(* CODESYS project Aufzug20.project

Project tree, tasks and I/O mapping:
  Device : CODESYS Control Win V3, 3S - Smart Software Solutions GmbH, order no. 305021, version 3.5.10.60
    application Application
      libraries: Standard, * (System); Util, * (System)
      task VISU_TASK (cyclic, interval 100 ms, priority 31) calls VisuElems.Visu_Prg
      task MainTask (cyclic, interval t#20ms, priority 1) calls PLC_PRG
      function block ManualControl [ST]
      data type Sensors
      global variables GVL_HMI
      global variables GVL_KONSTANTEN
      global variables GVL_AUFZUG
      Symbols
      program PLC_PRG [ST]
      function block OperatingMode [ST]
      visualisation Visualization
      function block DoorControl [ST]
      function SpeedCalculation [ST]
      function block Position [ST]
      function block MotorControl [ST]
      function block AuftragsTest [ST]
      data type Level
      function block LevelAnfahren [ST]
      function CalculateDirection [ST]
      function block Auftragsmanager [ST]
    Ethernet : Ethernet, 3S - Smart Software Solutions GmbH, version 3.5.10.0
        settings: IPAddress = [141,37,200,19]; SubnetMask = [255,255,255,255]; GatewayAddress = [0,0,0,0]; MACAddress = [16#00,16#00,16#00,16#00,16#00,16#00]; NetworkInterfaceName = 'htwg'; NetworkInterfaceName = "htwg"; SaveCommunicationSettings = FALSE
      Modbus_TCP_Master : Modbus TCP Master, 3S - Smart Software Solutions GmbH, version 3.5.10.0
        Modbus_TCP_Slave : Modbus TCP Slave, 3S - Smart Software Solutions GmbH, version 3.5.10.0
            settings: IPAddress = [141, 37, 159, 111]; Port = 503; Channel 0.Function Code = 4; Channel 0.Read Offset = 16#0000; Channel 0.Read Length = 7; Channel 0.Write Offset = 0; Channel 0.Write Length = 0; Channel 0.Cycle Time = 100; Channel 1.Function Code = 16; Channel 1.Read Offset = 0; Channel 1.Read Length = 0; Channel 1.Write Offset = 16#0000; Channel 1.Write Length = 2; Channel 1.Cycle Time = 100
            unmapped channels: Channel 0, Channel 1
  text list GlobalTextList
*)

// Device/Application/Sensors
TYPE Sensors :
STRUCT
	approach_lower :BOOL;
	safety_lower :BOOL;
	reached :BOOL;
	safety_upper :BOOL;
	approach_upper :BOOL;
END_STRUCT
END_TYPE

// Device/Application/Level
TYPE Level :
STRUCT
	sensors : Sensors;
	anforderungNachOben	: BOOL;
	anforderungNachUnten : BOOL;
END_STRUCT
END_TYPE

// Device/Application/GVL_HMI
{attribute 'qualified_only'}
VAR_GLOBAL
	//------------------------------------------------------------------------------------
	// Buttons
		// Operator								Taster die der Operator und Supervisor siehr
		Button_DoorClose			:BOOL;		// Taster innen Anforderung Tür schließen
		Button_DoorOpen				:BOOL;		// Taster innen Anforderung Türe Öffnen
		Button_EmergencyStop		:BOOL;		// Taster innen Anforderung Nothalt
		Buttons_level				:ARRAY[GVL_KONSTANTEN.min_level..GVL_KONSTANTEN.max_level] OF BOOL;
												// Taster innen Anforderung der Level (In unserem Fall Level 1,2,3,4)
		Buttons_Up					:ARRAY[GVL_KONSTANTEN.min_level..(GVL_KONSTANTEN.max_level-1)] OF BOOL;
												// Taster außen Anforderung Hochfahren (In unserem Fall Level 1,2,3)
		Buttons_Down				:ARRAY[(GVL_KONSTANTEN.min_level+1)..GVL_KONSTANTEN.max_level] OF BOOL;
												// Taster außen Anforderung Runterfahren (In unserem Fall Level 2,3,4)
												
		// Supervisor							Taster die der Supervisor zusätzlich hat
		Button_Reset				:BOOL;		// Taster Simulation-Reset
		Button_DoorCloseManual		:BOOL;		// Taster Handbetrieb Türe schließen
		Button_DoorOpenManual		:BOOL;		// Taster Handbetrieb Türe öffnen
		Button_MotorUpV1Manual		:BOOL;		// Taster Handbetrieb hochfahren mit V1
		Button_MotorUpV2Manual		:BOOL;		// Taster Handbetrieb hochfahren mit V2
		Button_MotorUpCrawlManual	:BOOL;		// Taster Handbetrieb hochfahren mit Kriechgeschwindigkeit
		Button_MotorDownV1Manual	:BOOL;		// Taster Handbetrieb runterfahren mit V1
		Button_MotorDownV2Manual	:BOOL;		// Taster Handbetrieb runterfahren mit V2
		Button_MotorDownCrawlManual	:BOOL;		// Taster Handbetrieb runterfahren mit Kriechgeschwindigkeit
		Button_AutomaticMode		:BOOL;		// Taster Anforderung Automatikmodus
		Button_ManualMode			:BOOL;		// Taster Anforderung Handbetrieb
		
		Button_deleteRequests		:BOOL;
		
		SupervisorActive			:BOOL;		// Variable Benutzerebenen
		
	//------------------------------------------------------------------------------------
	// Anzeigen
		ErrorState					:BOOL;		// Anzeige Aufzug befindet sich in Fehlerzustand
		
		DoorOpens					:BOOL;		// Anzeige Türe öffnet sich
		DoorCloses					:BOOL; 		// Anzeige Türe schließt sich
		DoorIsOpen					:BOOL;		// Anzeige Türe ist offen
		DoorIsClosed				:BOOL;		// Anzeige Türe ist geschlossen
		
		SimulationDoorIsOpen		:ARRAY[GVL_KONSTANTEN.min_level..GVL_KONSTANTEN.max_level] OF BOOL;
												// Simulation, welche Türe in welcher Etage offen ist
		
		AutomaticMode				:BOOL;		// Anzeige Automatikmodus
		ManualMode					:BOOL;		// Anzeige Handbetrieb
		
		MotorReady					:BOOL;		// Anzeige Motor ist bereit
		MotorOn						:BOOL;		// Anzeige Motor läuft
		MotorUp						:BOOL;		// Anzeige Aufzug fährt nach oben
		MotorDown					:BOOL;		// Anzeige Aufzug fährt nach unten
		MotorUpV1					:BOOL;		// Anzeige Aufzug fährt nach oben mit V1
		MotorUpV2					:BOOL;		// Anzeige Aufzug fährt nach oben mit V2
		MotorUpCrawl				:BOOL;		// Anzeige Aufzug fährt nach oben mit Kriechgeschwindigkeit
		MotorDownV1					:BOOL;		// Anzeige Aufzug fährt nach unten mit V1
		MotorDownV2					:BOOL;		// Anzeige Aufzug fährt nach unten mit V2
		MotorDownCrawl				:BOOL;		// Anzeige Aufzug fährt nach unten mit Kriechgeschwindigkeit
		Speed						:REAL;		// Anzeige akturelle Geschwindigkeit in m/s
		
		CurrentLevel				:INT;		// Anzeige in welchem Level sich der Aufzug gerade befindet
		TargetLevel					:INT;		// Anzeige, des aktuellen ZielStockwerks
		
		Requests					:ARRAY[GVL_KONSTANTEN.min_level..GVL_KONSTANTEN.max_level, 1..3] OF BOOL;
												// Anzeigen welche Stockwerke angefordert werden
		Sensors						:ARRAY[GVL_KONSTANTEN.min_level..GVL_KONSTANTEN.max_level, 1..5] OF BOOL;
												// Anzeige aktiver Sensoren
		LevelArrival				:ARRAY[GVL_KONSTANTEN.min_level..GVL_KONSTANTEN.max_level] OF BOOL;
		LevelDeparture				:ARRAY[GVL_KONSTANTEN.min_level..GVL_KONSTANTEN.max_level] OF BOOL;
		Position					:INT;		// Anzeige Aufzugsposition in mm
		
												
END_VAR

// Device/Application/GVL_KONSTANTEN
{attribute 'qualified_only'}
VAR_GLOBAL CONSTANT
	min_level	:INT:=1;
	max_level	:INT:=4;
	
	holding_period	:TIME:=T#6S;
END_VAR

// Device/Application/GVL_AUFZUG
{attribute 'qualified_only'}
VAR_GLOBAL
	// Ausgänge
	POreset 			AT %QX0.0 : BOOL; 		// Simulation reset
	POdv2 				AT %QX1.0 : BOOL; 		// motor setpoint down v2
	POdv1 				AT %QX1.1 : BOOL; 		// motor setpoint down v1
	POuv1 				AT %QX1.2 : BOOL; 		// motor setpoint up v1
	POuv2 				AT %QX1.3 : BOOL; 		// motor setpoint up v2
	POdclose 			AT %QX1.4 : BOOL; 		// motor close door
	POdopen 			AT %QX1.5 : BOOL; 		// motor open door
	POv_crawlSelect 	AT %QW1 : INT (-5..5); 	// select crawl speed; -5..5 cm/s
	
	// Eingänge
	PIs_l1sl 			AT %IX0.1 : BOOL; 		// Level 1 safety lower
	PIs_l1r 			AT %IX0.2 : BOOL; 		// Level 1 reached
	PIs_l1su 			AT %IX0.3 : BOOL; 		// Level 1 safety upper
	PIs_l1au 			AT %IX0.4 : BOOL; 		// Level 1 approach upper
	PIs_l2al 			AT %IX1.0 : BOOL; 		// Level 2 approach lower
	PIs_l2sl 			AT %IX1.1 : BOOL; 		// etc.
	PIs_l2r 			AT %IX1.2 : BOOL;
	PIs_l2su 			AT %IX1.3 : BOOL;
	PIs_l2au 			AT %IX1.4 : BOOL;
	PIs_l3al 			AT %IX2.0 : BOOL;
	PIs_l3sl 			AT %IX2.1 : BOOL;
	PIs_l3r 			AT %IX2.2 : BOOL;
	PIs_l3su 			AT %IX2.3 : BOOL;
	PIs_l3au 			AT %IX2.4 : BOOL;
	PIs_l4al 			AT %IX3.0 : BOOL;
	PIs_l4sl 			AT %IX3.1 : BOOL;
	PIs_l4r 			AT %IX3.2 : BOOL;
	PIs_l4su 			AT %IX3.3 : BOOL;
	PIcycles 			AT %ID1 : UDINT; 		// PLC cycles since start
	PIaufzugID 			AT %IW4 : UINT; 		// instance identifier (1..4)
	PIs_dopened 		AT %IX10.0 : BOOL; 		// door is open
	PIs_dclosed 		AT %IX10.1 : BOOL; 		// door is closed
	PIm_ready 			AT %IX10.2 : BOOL; 		// motor ready
	PIm_on 				AT %IX10.3 : BOOL; 		// motor is on
	PIm_error 			AT %IX10.4 : BOOL; 		// error state; reset with POreset
	PIs_v 				AT %IW6 : INT; 			// v [v]=1cm/s
END_VAR

// Device/Application/PLC_PRG
PROGRAM PLC_PRG
VAR	
	levels : ARRAY[GVL_KONSTANTEN.min_level..GVL_KONSTANTEN.max_level] OF Level;
	
	// FB Instanzen
	betriebsart			:OperatingMode;
	handBetrieb			:ManualControl;
	tuere  				: DoorControl;
	position 			: Position;
	motorControl 		: MotorControl;
	auftrag				: AuftragsTest;
	auftragsmanager		: Auftragsmanager;
	
	// Schnittstellen Funktionsbausteine
	automatik_ein				: BOOL;
	handbetrieb_ein				: BOOL;
	elevator_in_reached_position	: BOOL;
	level_target				: INT;
	level_current				: INT;
	level_target_reached		: BOOL;
	waiting_for_request			: BOOL;
	request_door_aut			: BOOL;

	// Zähler
	i : INT;
	
END_VAR

// Initialisierung Array
levels[GVL_KONSTANTEN.min_level].sensors.approach_lower		:= FALSE;
levels[GVL_KONSTANTEN.min_level].sensors.safety_lower		:= GVL_AUFZUG.PIs_l1sl;
levels[GVL_KONSTANTEN.min_level].sensors.reached			:= GVL_AUFZUG.PIs_l1r;
levels[GVL_KONSTANTEN.min_level].sensors.safety_upper		:= GVL_AUFZUG.PIs_l1su;
levels[GVL_KONSTANTEN.min_level].sensors.approach_upper		:= GVL_AUFZUG.PIs_l1au;
levels[GVL_KONSTANTEN.min_level].anforderungNachUnten		:= FALSE;
levels[GVL_KONSTANTEN.min_level].anforderungNachOben		:= GVL_HMI.Buttons_Up[GVL_KONSTANTEN.min_level];

levels[2].sensors.approach_lower							:= GVL_AUFZUG.PIs_l2al;
levels[2].sensors.safety_lower								:= GVL_AUFZUG.PIs_l2sl;
levels[2].sensors.reached									:= GVL_AUFZUG.PIs_l2r;
levels[2].sensors.safety_upper								:= GVL_AUFZUG.PIs_l2su;
levels[2].sensors.approach_upper							:= GVL_AUFZUG.PIs_l2au;
levels[2].anforderungNachUnten								:= GVL_HMI.Buttons_Down[2];
levels[2].anforderungNachOben								:= GVL_HMI.Buttons_Up[2];

levels[3].sensors.approach_lower							:= GVL_AUFZUG.PIs_l3al;
levels[3].sensors.safety_lower								:= GVL_AUFZUG.PIs_l3sl;
levels[3].sensors.reached									:= GVL_AUFZUG.PIs_l3r;
levels[3].sensors.safety_upper								:= GVL_AUFZUG.PIs_l3su;
levels[3].sensors.approach_upper							:= GVL_AUFZUG.PIs_l3au;
levels[3].anforderungNachUnten								:= GVL_HMI.Buttons_Down[3];
levels[3].anforderungNachOben								:= GVL_HMI.Buttons_Up[3];

levels[GVL_KONSTANTEN.max_level].sensors.approach_lower		:= GVL_AUFZUG.PIs_l4al;
levels[GVL_KONSTANTEN.max_level].sensors.safety_lower		:= GVL_AUFZUG.PIs_l4sl;
levels[GVL_KONSTANTEN.max_level].sensors.reached			:= GVL_AUFZUG.PIs_l4r;
levels[GVL_KONSTANTEN.max_level].sensors.safety_upper		:= GVL_AUFZUG.PIs_l4su;
levels[GVL_KONSTANTEN.max_level].sensors.approach_upper		:= FALSE;
levels[GVL_KONSTANTEN.max_level].anforderungNachUnten		:= GVL_HMI.Buttons_Down[GVL_KONSTANTEN.max_level];
levels[GVL_KONSTANTEN.max_level].anforderungNachOben		:= FALSE;

//------------------------------------------------------------------------------------
// Funktionsbausteine 

// Betriebsart 
betriebsart(
	wechsel_in_automatik := PLC_PRG.elevator_in_reached_position
	);
	
	automatik_ein:= PLC_PRG.betriebsart.automatikBetrieb;
	handbetrieb_ein:= PLC_PRG.betriebsart.handBetrieb;


// Handbetrieb
handBetrieb(
	enableManualControl := PLC_PRG.handbetrieb_ein, 
	freigabe_tuere:= PLC_PRG.elevator_in_reached_position
	);

// Positionsauswertung
position(
	levels:= PLC_PRG.levels
	);
	
	PLC_PRG.elevator_in_reached_position := position.elevator_in_reached_positon;
	PLC_PRG.level_current := position.level_current;

// Motorsteuerung Aufzug	
motorControl(
	automatic_mode := PLC_PRG.automatik_ein,
	levels := PLC_PRG.levels,
	reset := GVL_HMI.Button_Reset,
	level_target := PLC_PRG.level_target,
	level_current := PLC_PRG.level_current,
	emergency_stop := GVL_HMI.Button_EmergencyStop,
	request_DoorControl_start := GVL_HMI.Button_DoorOpen OR PLC_PRG.request_door_aut
	);
	
	PLC_PRG.waiting_for_request := motorControl.waiting_for_request;
	PLC_PRG.level_target_reached := motorControl.next_level_reached;

// Auftragsverarbeitung
auftrag(
	neuen_Auftrag_annehmen:= PLC_PRG.waiting_for_request
	);
	
	//level_target := auftrag.zielstockwerk;

// Auftragsmanager
auftragsmanager(
	levels := PLC_PRG.levels,
	buttons_inside := GVL_HMI.Buttons_level,
	level_current := PLC_PRG.level_current,
	level_target_reached := PLC_PRG.level_target_reached,
	waiting_for_request := PLC_PRG.waiting_for_request,
	request_door_aut	:= ,
	reset				:= GVL_HMI.Button_Reset
	);
	
	PLC_PRG.request_door_aut := auftragsmanager.request_door_aut;
	PLC_PRG.level_target := auftragsmanager.level_target;

// Ausgänge HMI - Anzeigen, Simulationen
GVL_HMI.AutomaticMode := automatik_ein;
GVL_HMI.ManualMode := handbetrieb_ein;

GVL_HMI.ErrorState := GVL_AUFZUG.PIm_error;

GVL_HMI.MotorUpV1 := GVL_AUFZUG.POuv1;
GVL_HMI.MotorUpV2 := GVL_AUFZUG.POuv2;
GVL_HMI.MotorUpCrawl := GVL_AUFZUG.POv_crawlSelect > 0;
GVL_HMI.MotorDownV1 := GVL_AUFZUG.POdv1;
GVL_HMI.MotorDownV2 := GVL_AUFZUG.POdv2;
GVL_HMI.MotorDownCrawl := GVL_AUFZUG.POv_crawlSelect < 0;
GVL_HMI.DoorCloses := GVL_AUFZUG.POdclose;
GVL_HMI.DoorOpens := GVL_AUFZUG.POdopen;
GVL_HMI.DoorIsClosed := GVL_AUFZUG.PIs_dclosed;
GVL_HMI.DoorIsOpen := GVL_AUFZUG.PIs_dopened;

GVL_HMI.MotorDown := motorControl.aufzug_faehrt_nach_unten;
GVL_HMI.MotorUp := motorControl.aufzug_faehrt_nach_oben;

GVL_HMI.CurrentLevel := level_current;
GVL_HMI.TargetLevel := level_target;

GVL_HMI.Requests := auftragsmanager.requests;
GVL_HMI.LevelArrival := motorControl.levelArrival;
GVL_HMI.LevelDeparture := motorControl.levelDeparture;


GVL_HMI.Speed := SpeedCalculation(GVL_AUFzug.PIs_v);
GVL_HMI.Position := position.position;

FOR i := GVL_KONSTANTEN.min_level TO GVL_KONSTANTEN.max_level BY 1 DO
	GVL_HMI.Sensors[i,1] := levels[i].sensors.approach_lower;
	GVL_HMI.Sensors[i,2] := levels[i].sensors.safety_lower;
	GVL_HMI.Sensors[i,3] := levels[i].sensors.reached;
	GVL_HMI.Sensors[i,4] := levels[i].sensors.safety_upper;
	GVL_HMI.Sensors[i,5] := levels[i].sensors.safety_upper;	
END_FOR

FOR i := GVL_KONSTANTEN.min_level TO GVL_KONSTANTEN.max_level BY 1 DO
	IF GVL_AUFZUG.PIs_dclosed THEN
		GVL_HMI.SimulationDoorIsOpen[i] := FALSE;
	END_IF
END_FOR

IF GVL_AUFZUG.PIs_dopened THEN
	GVL_HMI.SimulationDoorIsOpen[position.level_current] := TRUE;
END_IF

// Ausgänge Aufzug-Simulation
GVL_AUFZUG.POreset := GVL_HMI.Button_Reset;

GVL_AUFZUG.POuv1 := handbetrieb.MotorUpV1 OR motorControl.up_V1;
GVL_AUFZUG.POuv2 := handbetrieb.MotorUpV2 OR motorControl.up_V2;
GVL_AUFZUG.POdv1 := handbetrieb.MotorDownV1 OR motorControl.down_V1;
GVL_AUFZUG.POdv2 := handbetrieb.MotorDownV2 OR motorControl.down_V2;
IF handbetrieb_ein AND NOT automatik_ein THEN
	GVL_AUFZUG.POv_crawlSelect := handbetrieb.MotorCrawlSelect;
ELSIF automatik_ein AND NOT handbetrieb_ein THEN
	GVL_AUFZUG.POv_crawlSelect := motorControl.crawl_select;
END_IF
GVL_AUFZUG.POdopen := handbetrieb.MotorOpenDoor OR motorControl.door_open;
GVL_AUFZUG.POdclose := handbetrieb.MotorCloseDoor OR motorControl.door_close;

END_PROGRAM

// Device/Application/Position
FUNCTION_BLOCK Position
VAR_INPUT
	levels : ARRAY[GVL_KONSTANTEN.min_level..GVL_KONSTANTEN.max_level] OF Level;
END_VAR
VAR_OUTPUT
	elevator_in_reached_positon : BOOL;
	level_current : INT;
	position : INT;
	
	
END_VAR
VAR
	i : INT;
	postion_integral : INT;
	positon_sensor : INT;
	integral : INTEGRAL;
	resetIntegral : BOOL:=TRUE;
END_VAR

// Init
elevator_in_reached_positon := FALSE;

integral(
	IN:= GVL_AUFzug.PIs_v,
	TM:=20,
	RESET:= resetIntegral);

postion_integral := REAL_TO_INT(integral.OUT * 10);

resetIntegral:= FALSE;	

// Schleife
FOR i := GVL_KONSTANTEN.min_level TO GVL_KONSTANTEN.max_level BY 1 DO
	
	IF levels[i].sensors.reached THEN
		elevator_in_reached_positon:=TRUE;
		resetIntegral := TRUE;
		positon_sensor := i*3500 - 3500;
		level_current:= i;
	END_IF
	
	IF levels[i].sensors.approach_lower THEN
		resetIntegral := TRUE;
		positon_sensor := i*3500 - 3500 - 1500;
		level_current:= i;
	END_IF
	
	IF levels[i].sensors.safety_lower THEN
		resetIntegral := TRUE;
		positon_sensor := i*3500 -3500 -50;
		level_current:= i;
	END_IF
	
	IF levels[i].sensors.safety_upper THEN
		resetIntegral := TRUE;
		positon_sensor := i*3500 - 3500 + 50;
		level_current:= i;
	END_IF
	
	IF levels[i].sensors.approach_upper THEN
		resetIntegral := TRUE;
		positon_sensor := i*3500 -3500 + 1500;
		level_current:= i;
	END_IF
	
END_FOR

// Ausgänge
position := positon_sensor + postion_integral;

END_FUNCTION_BLOCK

// Device/Application/MotorControl
FUNCTION_BLOCK MotorControl
VAR_INPUT
	levels 				: ARRAY[GVL_KONSTANTEN.min_level..GVL_KONSTANTEN.max_level] OF Level;
	reset 				: BOOL;
	level_target 		: INT := GVL_KONSTANTEN.min_level;
	level_current 		: INT := GVL_KONSTANTEN.max_level;
	automatic_mode 		: BOOL;
	emergency_stop 		: BOOL;
	request_DoorControl_start 	: BOOL;
END_VAR
VAR_OUTPUT
	up_V1 : BOOL;
	up_V2 : BOOL;
	down_V1 : BOOL;
	down_V2 : BOOL;
	crawl_select : INT;
	door_open : BOOL;
	door_close : BOOL;
	
	waiting_for_request : BOOL;
	next_level_reached : BOOL;
	
	levelArrival				:ARRAY[GVL_KONSTANTEN.min_level..GVL_KONSTANTEN.max_level] OF BOOL;
	levelDeparture				:ARRAY[GVL_KONSTANTEN.min_level..GVL_KONSTANTEN.max_level] OF BOOL;
	
	aufzug_faehrt_nach_oben : BOOL;
	aufzug_faehrt_nach_unten : BOOL;
END_VAR
VAR
	z		: INT:=0;
	
	direction_up : BOOL; 
	direction_down : BOOL;
	
	levelAnfahrenNachOben	: LevelAnfahren;
	levelAnfahrenNachUnten	: LevelAnfahren;
	doorControl : DoorControl;
END_VAR

levelAnfahrenNachOben(
	start := (z=20),
	sensor_reached := levels[level_target].sensors.reached,
	sensor_safty_before := levels[level_target].sensors.safety_lower,
	sensor_safty_after := levels[level_target].sensors.safety_upper,
	sensor_approach := levels[level_target].sensors.approach_lower,
	emergency_stop := emergency_stop,
	reset := reset OR NOT automatic_mode,
	direction_up := TRUE
	);
	
levelAnfahrenNachUnten(
	start := (z=30),
	sensor_reached := levels[level_target].sensors.reached,
	sensor_safty_before := levels[level_target].sensors.safety_upper,
	sensor_safty_after := levels[level_target].sensors.safety_lower,
	sensor_approach := levels[level_target].sensors.approach_upper,
	emergency_stop := emergency_stop,
	reset := reset OR NOT automatic_mode,
	direction_up := FALSE
	);

doorControl(
	aut_start:= z=40
	);

// Gehe in Initialisierungszustand, wenn Reset
IF reset OR NOT automatic_mode THEN
	z:=0;
	direction_up :=FALSE;
	direction_down := FALSE;
END_IF 

// Zustandsautomat
CASE z OF
	// Init, Reset
	0:
	IF GVL_AUFZUG.PIm_ready THEN
		z:=10;
	END_IF
	
	// Wartezustand - Aufzug befindet sich in Ziellevel und wartet auf nächsten Auftrag
	10:
	IF level_target > level_current THEN
		z:=20;
	ELSIF level_target < level_current THEN
		z:= 30;
	END_IF
	
	IF request_DoorControl_start THEN
		z:= 40;
	END_IF
	
	// Impuls nach oben Anfahren
	20:
	z:= 21;
	
	//  Level anfahren
	21:
	IF levelAnfahrenNachOben.level_reached THEN
		z:=40;
	END_IF
	
	// Impuls nach unten Anfahren
	30:
	z:= 31;
	
	// Level Anfahren
	31:
	IF levelAnfahrenNachUnten.level_reached THEN
		z:=40;
	END_IF
	
	// Impuls Türautomatik Start, Level Angefahren
	40:
	z:= 41;
	
	// Warte auf Ende Türautomatik	
	41:
	IF doorControl.aut_ende THEN
		z:=10;
	END_IF
	
END_CASE
	

up_V1 := levelAnfahrenNachOben.v1;
up_V2 := levelAnfahrenNachOben.v2;
down_V1 := levelAnfahrenNachUnten.v1;
down_V2 := levelAnfahrenNachUnten.v2;
door_open := doorControl.door_open;
door_close := doorControl.door_close;

IF levelAnfahrenNachOben.fb_active THEN
	crawl_select := levelAnfahrenNachOben.crawl_select;
ELSIF levelAnfahrenNachUnten.fb_active THEN
	crawl_select := levelAnfahrenNachUnten.crawl_select;
ELSE
	crawl_select := 0;
END_IF

waiting_for_request := z=10 OR z=40 OR z=41;
next_level_reached := z=40;

IF z=10 OR z=40 OR z=41 THEN
	levelArrival[level_current] := TRUE;
ELSE
	levelArrival[level_current] := FALSE;
END_IF
IF z=20 OR z=30 THEN
	levelDeparture[level_current] :=TRUE;
ELSE
	levelDeparture[level_current] :=FALSE;
END_IF

aufzug_faehrt_nach_oben := levelAnfahrenNachOben.fb_active;
aufzug_faehrt_nach_unten := levelAnfahrenNachUnten.fb_active;

END_FUNCTION_BLOCK

// Device/Application/DoorControl
FUNCTION_BLOCK DoorControl
VAR_INPUT
	aut_start : BOOL;
END_VAR
VAR_OUTPUT
	aut_ende :BOOL;
	door_open : BOOL;
	door_close : BOOL;
END_VAR
VAR
	z: INT:=0;
	ton_halten :TON;
	i_max : INT:=3;
END_VAR

ton_halten(IN:=z=3, PT:= T#6S);

CASE z OF
	// Init
	0:
	z:=1;
	
	// Wartezustand
	1:
	IF aut_start  THEN
		z:=2;
		i_max:=3;
	END_IF
	
	// Tuere öffnen
	2:
	IF GVL_AUFZUG.PIs_dopened THEN
		z:=3;
	END_IF
	
	// Tuere offen halten
	3:
	IF ton_halten.Q OR GVL_HMI.Button_DoorCloseManual OR GVL_HMI.Button_DoorClose THEN
		z:=4;
	END_IF
	
	// Tuere schließen
	4:
	IF GVL_AUFZUG.PIs_dclosed THEN
		z:=5;
	END_IF
	IF i_max > 0 AND (GVL_HMI.Button_DoorOpenManual OR GVL_HMI.Button_DoorOpen) THEN			// Türe wieder aufmachen
		z:=2;
		i_max:= i_max - 1;
	END_IF
	
	// Ende
	5:
	z:=0;
END_CASE

// Ausgänge
aut_ende := z=5;
door_open:= z=2;
door_close:= z=4;

END_FUNCTION_BLOCK

// Device/Application/LevelAnfahren
FUNCTION_BLOCK LevelAnfahren
VAR_INPUT
	start 				: BOOL;
	sensor_reached 		: BOOL;
	sensor_safty_before : BOOL;
	sensor_safty_after	: BOOL;
	sensor_approach		: BOOL;
	emergency_stop		: BOOL;
	reset				: BOOL;
	direction_up		: BOOL;
END_VAR
VAR_OUTPUT
	v1	: BOOL;
	v2 	: BOOL;
	crawl_select	: INT :=0;
	level_reached	: BOOL;
	fb_active		: BOOL;
END_VAR
VAR
	z					: INT :=0;
	
	ton_V1				: TON;
	ton_V2				: TON;
	ton_check_reached	: TON;
	
	sensor_approach_ausgeloest		: BOOL;
	sensor_safty_before_ausgeloest	: BOOL;
	
	multiplicator	: INT:=1;
	
END_VAR

// Zeitglieder initialisieren
ton_V1(IN:= (z=3), PT:= T#1S);
ton_V2(IN:= (z=2), PT:= T#0.1S);
ton_check_reached(IN:= (z=6), PT:= T#0.5S);

IF reset THEN
	z:= 0;
END_IF

IF emergency_stop AND (z<>0) THEN
	z:= 99;
END_IF

IF sensor_approach THEN
	sensor_approach_ausgeloest :=TRUE;
END_IF

IF sensor_safty_before THEN
	sensor_safty_before_ausgeloest := TRUE;
END_IF

IF direction_up THEN
	multiplicator := 1;
ELSE
	multiplicator := -1;
END_IF

CASE z OF
	// Init, Reset, Automatikmodus aus
	0:
	sensor_approach_ausgeloest 		:= FALSE;
	sensor_safty_before_ausgeloest 	:= FALSE;
	
	IF start THEN
		z:=1;
	END_IF
	
	// Fahre mit V2 bis Zielstockwerk sich nähert
	1:
	IF sensor_approach THEN
		z:=2;
	END_IF
	
	// Verzögerung, weiter mit V2 - Optimierung der Fahrzeit
	2:
	IF ton_v2.Q THEN
		z:=3;
	END_IF
	
	// Fahre mit V1 bis korrekte Position sich nähert
	3:
	IF ton_v1.Q THEN
		z:=4;
	END_IF
	
	// Fahre mit Kriechgeschwindigkeit 4 
	4:
	IF sensor_safty_before THEN
		z:=5;
	END_IF
	
	// Fahre mit Kriechgeschwindigkeit 1
	5:
	IF sensor_reached THEN
		z:=6;
	END_IF
	
	// Prüfe ob lange genug in reach Position
	6:
	IF ton_check_reached.Q AND sensor_reached THEN
		z:=10;
	ELSIF (ton_check_reached.Q AND NOT sensor_reached) OR sensor_safty_after THEN
		z:=7;
	END_IF
	
	// Fahre mit Kriechgeschwindigkeit Stockwerk korrekt an
	7:
	IF sensor_reached THEN
		z:=6;
	END_IF
	
	// Stockwerk erreicht
	10:
	z:=0;
	
	// Nothalt
	99:
	IF NOT emergency_stop THEN
		IF sensor_approach_ausgeloest AND NOT sensor_safty_before_ausgeloest THEN
			z:=4;
		ELSIF sensor_safty_before_ausgeloest THEN
			z:=5;
		ELSE
			z:=1;
		END_IF
	END_IF
	
END_CASE


// Ausgänge setzen
v1	:= (z=3);
v2	:= (z=1 OR z=2);

CASE z OF
	4:
	crawl_select :=4 * multiplicator;
	5:
	crawl_select := 1 * multiplicator;
	6:
	crawl_select := -1 * multiplicator;
ELSE
	crawl_select := 0;
END_CASE

level_reached := (z=10);
fb_active := z<>0;

END_FUNCTION_BLOCK

// Device/Application/Auftragsmanager
FUNCTION_BLOCK Auftragsmanager
VAR_INPUT
	levels : ARRAY[GVL_KONSTANTEN.min_level..GVL_KONSTANTEN.max_level] OF Level;
	buttons_inside : ARRAY[GVL_KONSTANTEN.min_level..GVL_KONSTANTEN.max_level] OF BOOL;
	level_current	: INT;
	level_target_reached	: BOOL;
	waiting_for_request	: BOOL;
	reset : BOOL;
END_VAR
VAR_OUTPUT
	level_target	: INT := GVL_KONSTANTEN.min_level;
	requests : ARRAY[GVL_KONSTANTEN.min_level..GVL_KONSTANTEN.max_level, 1..3] OF BOOL;
	request_door_aut	: BOOL;
END_VAR
VAR
	i : INT;
	j : INT;
	z : INT:=0;	
	ton_waitingUP				: TON;
	ton_waitingDOWN				: TON;
	requestsAvailableUp : BOOL;
	requestsAvailableUpOverLevelCurrent : BOOL;
	requestsAvailableUpUnderLevelCurrent : BOOL;
	requestsAvailableDown : BOOL;
	requestsAvailableDownOverLevelCurrent : BOOL;
	requestsAvailableDownUnderLevelCurrent : BOOL;
END_VAR

// Anforderungen annehmen
FOR i := GVL_KONSTANTEN.min_level TO GVL_KONSTANTEN.max_level BY 1 DO
	IF levels[i].anforderungNachOben THEN									// Außen nach Oben [level,1]
		requests[i,1] := TRUE;
	END_IF
	IF levels[i].anforderungNachUnten THEN
		requests[i,2] := TRUE;												// Außen nach Unten [level,2]
	END_IF
	IF buttons_inside[i] AND i <> level_current THEN
		requests[i,3] := TRUE;												// Innen [level,3]
	END_IF
END_FOR


// Alle Anforderungen löschen und in unterstes Level fahren
IF GVL_HMI.Button_deleteRequests OR reset THEN
	FOR i := GVL_KONSTANTEN.min_level TO GVL_KONSTANTEN.max_level BY 1 DO
		requests[i,1] := FALSE;
		requests[i,2] := FALSE;
		requests[i,3] := FALSE;
	END_FOR
	z:=0;
	level_target := GVL_KONSTANTEN.min_level;
END_IF

// Zeitglieder für Timeouts
ton_waitingUP(IN:= z=11, PT:=T#11S);
ton_waitingDOWN(IN:= z=21, PT:=T#11S);

CASE z OF
	// Wartezustand - Keine Aufträge vorhanden
	0:
	IF CalculateDirection(requests, level_current)= 10 THEN			// Anforderung von außen gleiches Stockwerk nach oben
		z:=10;
	END_IF
	IF CalculateDirection(requests, level_current)= -10 THEN		// Anforerung von außen gleiches Stockwerk nach unten
		z:=20;
	END_IF
	IF CalculateDirection(requests, level_current)= 1 THEN			// Anforderung von außen anderes Stockwerk nach oben
		z:=30;
	END_IF
	IF CalculateDirection(requests, level_current)= -1 THEN			// Anforderung von außen anderes Stockwerk nach unten
		z:=40;
	END_IF
	
	// Anforderung von Außen gleiches Stockwerk nach oben, Impuls Türe auf
	10:
	IF waiting_for_request THEN										// MotorControl bereit für Türoffnung
		z:=11;
	END_IF
	
	// Auftrag löschen
	11:
	requests[level_current,1] := FALSE;								// Anforderung gleiches Stockwerk nach oben löschen
	IF ton_waitingUP.Q THEN											// Timeout wenn im Aufzug nichts gedruckt wird (z.B. wenn keine Person eingestiegen ist
		z:=0;
	END_IF
	IF CalculateDirection(requests, level_current)=1 THEN			// Anforderung Richtung nach oben
		z:=30;
	END_IF
	
	// Anforderung von Außen gleiches Stockwerk nach unten, Impuls Türe auf, Auftrag löschen
	20:
	IF waiting_for_request THEN										// MotorControl bereit für Türoffnung
		z:=21;
	END_IF
	
	// Auftrag löschen
	21:
	requests[level_current,2] := FALSE;								// Anforderung gleiches Stockwerk nach unten löschen
	IF ton_waitingDOWN.Q THEN
		z:=0;
	END_IF
	IF CalculateDirection(requests, level_current)= -1 THEN			// Auftrag Richtung nach unten
		z:=40;
	END_IF
	
	// Berechne neues Zielstockwerk Fahrtrichtung aufwärts überhalb
	30:
	IF level_target_reached OR waiting_for_request THEN									// Auftrag löschen wenn in neuem Stockwerk angekommen
		requests[level_current,1] := FALSE;
		requests[level_current,3] := FALSE;
	END_IF
	
	IF  requestsAvailableDownUnderLevelCurrent AND (NOT requestsAvailableUpOverLevelCurrent) THEN
		IF waiting_for_request OR level_target_reached  THEN
			z:= 40;
			requests[level_current,3] := FALSE;
		END_IF
	END_IF
	
	
	IF (NOT requestsAvailableUpOverLevelCurrent) AND requestsAvailableUpUnderLevelCurrent THEN
		IF waiting_for_request OR level_target_reached  THEN
			z:= 31;
			requests[level_current,3] := FALSE;
		END_IF
	END_IF
	
	IF requests[level_current,1] THEN								// Anforderung von Außen gleiches Stockwerk nach oben -> Zustand 10
		z:=10;
	END_IF
	
	IF NOT (requestsAvailableUp OR  requestsAvailableDown) THEN		// Wenn keine Anforderungen mehr vorhanden sind gehe in Zustand 0
		requests[level_current,1] := FALSE;
		requests[level_current,3] := FALSE;
		z:=0;
	END_IF
	
	FOR i := GVL_KONSTANTEN.min_level TO GVL_KONSTANTEN.max_level BY 1 DO		// Berechne nächstes Zielstockwerk Fahrtrichtung nach oben
		IF (requests[i,1] OR requests[i,3]) AND i >= level_current THEN
			level_target := i;
			EXIT;
		END_IF
	END_FOR
	
	// Berechne neues Zielstockwerk Fahrtrichtung aufwärts unterhalb
	31:
	FOR i := GVL_KONSTANTEN.min_level TO GVL_KONSTANTEN.max_level BY 1 DO		// Berechne nächstes Zielstockwerk Fahrtrichtung nach oben
		IF (requests[i,1] OR requests[i,3]) AND i < level_current THEN
			level_target := i;
			EXIT;
		END_IF
	END_FOR
	
	IF level_target_reached OR waiting_for_request THEN
		requests[level_current,1] := FALSE;
		requests[level_current,3] := FALSE;
		z:=30;
	END_IF
	
	// Berechne neues Zielstockwerk Fahrtrichtung abwärts unterhalb
	40:
	IF level_target_reached OR waiting_for_request THEN									// Auftrag löschen wenn in neuem Stockwerk angekommen
		requests[level_current,2] := FALSE;
		requests[level_current,3] := FALSE;
	END_IF
	
	IF  requestsAvailableUpOverLevelCurrent AND (NOT requestsAvailableDownUnderLevelCurrent) THEN
		IF waiting_for_request OR level_target_reached  THEN
			requests[level_current,2] := FALSE;
			requests[level_current,3] := FALSE;
			z:= 30;
		END_IF
	END_IF
	
	
	IF (NOT requestsAvailableDownUnderLevelCurrent) AND requestsAvailableDownOverLevelCurrent THEN
		IF waiting_for_request OR level_target_reached  THEN
			requests[level_current,2] := FALSE;
			requests[level_current,3] := FALSE;
			z:= 41;
		END_IF
	END_IF
	
	IF requests[level_current,2] THEN								// Anforderung von Außen gleiches Stockwerk nach unten -> Zustand 10
		z:=10;
	END_IF
	
	IF NOT (requestsAvailableUp OR  requestsAvailableDown) THEN		// Wenn keine Anforderungen mehr vorhanden sind gehe in Zustand 0
		requests[level_current,2] := FALSE;
		requests[level_current,3] := FALSE;
		z:=0;
	END_IF
	
	FOR i := GVL_KONSTANTEN.max_level TO GVL_KONSTANTEN.min_level BY -1 DO		// Berechne nächstes Zielstockwerk Fahrtrichtung nach oben
		IF (requests[i,2] OR requests[i,3]) AND i <= level_current THEN
			level_target := i;
			EXIT;
		END_IF
	END_FOR
	
	
	//Berechne neues Zielstockwerk Fahrtrichtung abwärts überhalb
	41:
	FOR i := GVL_KONSTANTEN.max_level TO GVL_KONSTANTEN.min_level BY -1 DO		// Berechne nächstes Zielstockwerk Fahrtrichtung nach unten
		IF (requests[i,2] OR requests[i,3]) AND i > level_current THEN
			level_target := i;
			EXIT;
		END_IF
	END_FOR
	
	IF level_target_reached OR waiting_for_request THEN
		requests[level_current,2] := FALSE;
		requests[level_current,3] := FALSE;
		z:=40;
	END_IF
	
	
	
END_CASE

// Prüfe in welche Richtung Anforderungen vorhanden sind
requestsAvailableUp := FALSE;
requestsAvailableDown := FALSE;
requestsAvailableUpOverLevelCurrent := FALSE;
requestsAvailableUpUnderLevelCurrent := FALSE;
requestsAvailableDownOverLevelCurrent := FALSE;
requestsAvailableDownUnderLevelCurrent := FALSE;

FOR i := GVL_KONSTANTEN.min_level TO GVL_KONSTANTEN.max_level BY 1 DO
	IF requests[i,1] THEN
		requestsAvailableUp := TRUE;
		IF i > level_current THEN
			requestsAvailableUpOverLevelCurrent := TRUE;
		END_IF
		IF i < level_current THEN
			requestsAvailableUpUnderLevelCurrent := TRUE;
		END_IF
	END_IF
	IF requests[i,2] THEN
		requestsAvailableDown := TRUE;
		IF i > level_current THEN
			requestsAvailableDownOverLevelCurrent := TRUE;
		END_IF
		IF i< level_current THEN
			requestsAvailableDownUnderLevelCurrent := TRUE;
		END_IF
	END_IF
	IF requests[i,3] AND i < level_current  THEN
		requestsAvailableDown := TRUE;
		requestsAvailableUpUnderLevelCurrent := TRUE;
		requestsAvailableDownUnderLevelCurrent := TRUE;
	ELSIF requests[i,3] AND i > level_current THEN
		requestsAvailableUp := TRUE;
		requestsAvailableUpOverLevelCurrent := TRUE;
		requestsAvailableDownOverLevelCurrent := TRUE;
	END_IF
END_FOR

// Rücksetzen Anfordrung ganz oben und ganz unten
IF level_current=GVL_KONSTANTEN.max_level THEN
	requests[GVL_KONSTANTEN.max_level,2] := FALSE;
END_IF

IF level_current=GVL_KONSTANTEN.min_level THEN
	requests[GVL_KONSTANTEN.max_level,1] := FALSE;
END_IF

// Ausgänge setzen
request_door_aut := z=10 OR z=20;

END_FUNCTION_BLOCK

// Device/Application/CalculateDirection
FUNCTION CalculateDirection : INT
VAR_INPUT
	requests : ARRAY[GVL_KONSTANTEN.min_level..GVL_KONSTANTEN.max_level, 1..3] OF BOOL;
	level_current	: INT;
END_VAR
VAR
	i,j : INT:=0;
	value : INT := 99;
END_VAR

FOR i := GVL_KONSTANTEN.min_level TO GVL_KONSTANTEN.max_level BY 1 DO
	// Nach unten, gleiches Level
	IF requests[i,2] AND i = level_current THEN
		value := -10;
	END_IF
	// Nach oben, gleiches Level
	IF requests[i,1] AND i = level_current THEN
		value := 10;
	END_IF
	// Nach unten von außen
	IF (requests[i,2] AND i <> level_current) THEN
		value := -1;
	END_IF
	// Nach oben von außen
	IF requests[i,1] AND i <> level_current THEN
		value := 1;
	END_IF
	// Nach unten von innen
	IF requests[i,3] AND i < level_current THEN
		value :=- 1;
	END_IF
	//Nach oben von innen
	IF requests[i,3] AND i > level_current THEN
		value := 1;
	END_IF
END_FOR

CalculateDirection := value;

END_FUNCTION

// Device/Application/SpeedCalculation
FUNCTION SpeedCalculation : REAL
VAR_INPUT
	speed_cm_per_seconds : INT;
END_VAR
VAR
END_VAR

SpeedCalculation:= speed_cm_per_seconds / 100.0; // gibt die Fahrstuhlgeschwindigkeit in Meter pro Sekunde zurück

END_FUNCTION

// Device/Application/OperatingMode
FUNCTION_BLOCK OperatingMode
VAR_INPUT
	wechsel_in_automatik : BOOL;
END_VAR
VAR_OUTPUT
	automatikBetrieb: BOOL;
	handBetrieb: BOOL;
END_VAR
VAR
	z:INT:=0;
END_VAR

CASE z OF
	// Automatikbetrieb
	0:
	IF GVL_HMI.Button_ManualMode AND GVL_HMI.SupervisorActive THEN 
	z:=10;
	END_IF
	
	// Handbetrieb - wechsel in Automatikbetrieb nur möglich wenn 
	// Aufzug nicht in Fehlerzustand, der Motor nicht läuft, Supervisor aktiv 
	// der Aufzug im Hanbetrieb ein Stockwerk korrekt angefahren hat
	10:
	IF GVL_HMI.Button_AutomaticMode AND NOT GVL_AUFZUG.PIm_error AND NOT GVL_AUFZUG.PIm_on AND GVL_HMI.SupervisorActive AND wechsel_in_automatik THEN
	z:=0;
	END_IF
	
END_CASE

// Ausgänge
automatikBetrieb:= z=0;
handBetrieb:= z=10;

END_FUNCTION_BLOCK

// Device/Application/ManualControl
FUNCTION_BLOCK ManualControl
VAR_INPUT
	enableManualControl: BOOL;
	freigabe_tuere : BOOL;
END_VAR
VAR_OUTPUT
	MotorUpV1 : BOOL;
	MotorUpV2 : BOOL;
	MotorDownV1 : BOOL;
	MotorDownV2 : BOOL;
	
	MotorOpenDoor : BOOL;
	MotorCloseDoor : BOOL;
	
	MotorCrawlSelect : INT;
END_VAR
VAR
	MotorCloseDooer: BOOL;
END_VAR

MotorUpV1 := enableManualControl AND GVL_HMI.Button_MotorUpV1Manual AND GVL_AUFZUG.PIs_dclosed;
MotorUpV2 := enableManualControl AND GVL_HMI.Button_MotorUpV2Manual AND GVL_AUFZUG.PIs_dclosed;

MotorDownV1 := enableManualControl AND GVL_HMI.Button_MotorDownV1Manual AND GVL_AUFZUG.PIs_dclosed;
MotorDownV2 := enableManualControl AND GVL_HMI.Button_MotorDownV2Manual AND GVL_AUFZUG.PIs_dclosed;

MotorOpenDoor := enableManualControl AND GVL_HMI.Button_DoorOpenManual AND freigabe_tuere;
MotorCloseDoor := enableManualControl AND GVL_HMI.Button_DoorCloseManual AND freigabe_tuere;

IF enableManualControl AND GVL_AUFZUG.PIs_dclosed THEN
	IF GVL_HMI.Button_MotorDownCrawlManual THEN
		MotorCrawlSelect := -1;
	ELSIF GVL_HMI.Button_MotorUpCrawlManual THEN
		MotorCrawlSelect := 1;
	ELSE
		MotorCrawlSelect :=0;
	END_IF
END_IF

END_FUNCTION_BLOCK

// Device/Application/AuftragsTest
FUNCTION_BLOCK AuftragsTest
VAR_INPUT
	neuen_Auftrag_annehmen : BOOL;
END_VAR
VAR_OUTPUT
	zielstockwerk : INT:=GVL_KONSTANTEN.min_level;
END_VAR
VAR
	i : INT;
END_VAR

IF GVL_HMI.Button_Reset THEN
	zielstockwerk := GVL_KONSTANTEN.min_level;
END_IF

FOR i := GVL_KONSTANTEN.min_level TO GVL_KONSTANTEN.max_level BY 1 DO
	IF GVL_HMI.Buttons_level[i] AND neuen_Auftrag_annehmen THEN
		zielstockwerk := i;
	END_IF
END_FOR

END_FUNCTION_BLOCK

// Device/Application/Visualization
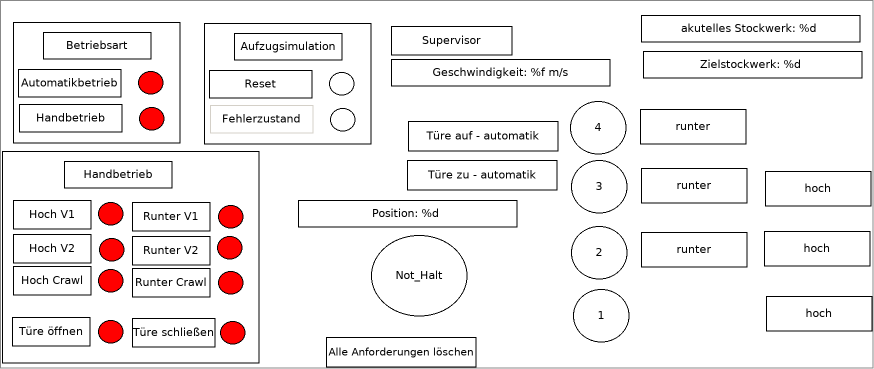
VISUALIZATION Visualization  // 874x369
    RoundedRectangle (13,22 167x121)
    RoundedRectangle (43,32 108x27), "Betriebsart"
    Rectangle (18,69 103x28), "Automatikbetrieb"
        tap GVL_HMI.Button_AutomaticMode
    Rectangle (19,104 103x28), "Handbetrieb"
        tap GVL_HMI.Button_ManualMode
    Ellipse (138,71 25x23), colour toggle: GVL_HMI.AutomaticMode
    Ellipse (139,107 25x23), colour toggle: GVL_HMI.ManualMode
    RoundedRectangle (204,23 167x121)
    RoundedRectangle (234,33 108x27), "Aufzugsimulation"
    Rectangle (209,70 103x28), "Reset"
        tap GVL_HMI.Button_Reset
    RoundedRectangle (210,105 103x28), "Fehlerzustand"
    Ellipse (329,72 25x23), colour toggle: GVL_HMI.Button_Reset
    Ellipse (330,108 25x23), colour toggle: GVL_HMI.ErrorState
    RoundedRectangle (2,151 257x212)
    RoundedRectangle (64,161 108x27), "Handbetrieb"
    Rectangle (13,200 78x29), "Hoch V1"
        tap GVL_HMI.Button_MotorUpV1Manual
    Rectangle (13,234 78x29), "Hoch V2"
        tap GVL_HMI.Button_MotorUpV2Manual
    Rectangle (13,266 78x29), "Hoch Crawl"
        tap GVL_HMI.Button_MotorUpCrawlManual
    Rectangle (132,202 78x29), "Runter V1"
        tap GVL_HMI.Button_MotorDownV1Manual
    Rectangle (132,236 78x29), "Runter V2"
        tap GVL_HMI.Button_MotorDownV2Manual
    Rectangle (132,268 78x29), "Runter Crawl"
        tap GVL_HMI.Button_MotorDownCrawlManual
    Rectangle (12,317 78x29), "Türe öffnen"
        tap GVL_HMI.Button_DoorOpenManual
    Rectangle (132,318 83x29), "Türe schließen"
        tap GVL_HMI.Button_DoorCloseManual
    Ellipse (98,202 25x23), colour toggle: GVL_HMI.MotorUpV1
    Ellipse (99,238 25x23), colour toggle: GVL_HMI.MotorUpV2
    Ellipse (98,269 25x23), colour toggle: GVL_HMI.MotorUpCrawl
    Ellipse (218,205 25x23), colour toggle: GVL_HMI.MotorDownV1
    Ellipse (217,236 25x23), colour toggle: GVL_HMI.MotorDownV2
    Ellipse (218,271 25x23), colour toggle: GVL_HMI.MotorDownCrawl
    Ellipse (98,320 25x23), colour toggle: GVL_HMI.DoorOpens
    Ellipse (220,321 25x23), colour toggle: GVL_HMI.DoorCloses
    Rectangle (391,26 121x29), "Supervisor"
        toggle GVL_HMI.SupervisorActive
    Rectangle (391,59 219x27), "Geschwindigkeit: %f m/s", text variable: GVL_HMI.Speed
    Ellipse (371,235 96x81), "Not_Halt"
        toggle GVL_HMI.Button_EmergencyStop
    Ellipse (573,289 56x53), "1", colour toggle: GVL_HMI.Requests[1,3]
        tap GVL_HMI.Buttons_level[1]
    Ellipse (571,226 56x53), "2", colour toggle: GVL_HMI.Requests[2,3]
        tap GVL_HMI.Buttons_level[2]
    Ellipse (571,160 56x53), "3", colour toggle: GVL_HMI.Requests[3,3]
        tap GVL_HMI.Buttons_level[3]
    Ellipse (570,101 56x53), "4", colour toggle: GVL_HMI.Requests[4,3]
        tap GVL_HMI.Buttons_level[4]
    Rectangle (408,121 150x30), "Türe auf - automatik"
        tap GVL_HMI.Button_DoorOpen
    Rectangle (407,160 150x30), "Türe zu - automatik"
        tap GVL_HMI.Button_DoorClose
    Rectangle (640,109 106x35), "runter", colour toggle: GVL_HMI.Requests[4,2]
        tap GVL_HMI.Buttons_Down[4]
    Rectangle (641,168 106x35), "runter", colour toggle: GVL_HMI.Requests[3,2]
        tap GVL_HMI.Buttons_Down[3]
    Rectangle (641,232 106x35), "runter", colour toggle: GVL_HMI.Requests[2,2]
        tap GVL_HMI.Buttons_Down[2]
    Rectangle (765,171 106x35), "hoch", colour toggle: GVL_HMI.Requests[3,1]
        tap GVL_HMI.Buttons_Up[3]
    Rectangle (764,231 106x35), "hoch", colour toggle: GVL_HMI.Requests[2,1]
        tap GVL_HMI.Buttons_Up[2]
    Rectangle (766,296 106x35), "hoch", colour toggle: GVL_HMI.Requests[1,1]
        tap GVL_HMI.Buttons_Up[1]
    Rectangle (641,15 219x27), "akutelles Stockwerk: %d", text variable: GVL_HMI.CurrentLevel
    Rectangle (643,51 219x27), "Zielstockwerk: %d", text variable: GVL_HMI.TargetLevel
    Rectangle (298,200 219x27), "Position: %d", text variable: GVL_HMI.Position
    Rectangle (326,337 150x30), "Alle Anforderungen löschen"
        tap GVL_HMI.Button_deleteRequests
END_VISUALIZATION
